// TIA Portal V17 export
// export: Created 2026-04-13T11:12:44.4398568Z, ExportSetting WithDefaults, DisplayName Totally Integrated Automation Portal, DisplayVersion V17 Update 4, DisplayName TIA Portal Openness, DisplayVersion V17 Update 4, DisplayName TIA Portal Version Control Interface, DisplayVersion V17, DisplayName SINAMICS Startdrive Advanced, DisplayVersion V17, DisplayName SINAMICS Startdrive G130, G150, S120, S150, SINAMICS MV, S210, DisplayVersion V17, DisplayName SINAMICS Startdrive G110M, G120, G120C, G120D, G120P, G115D, DisplayVersion V17, DisplayName STEP 7 Professional, DisplayVersion V17 Update 4, DisplayName STEP 7 Safety, DisplayVersion V17, DisplayName WinCC Professional, DisplayVersion V17 Update 4
DATA_BLOCK "6-ALLALARM_DB"   // DB23
VERSION : 0.1
// stored: AutoNumber true, DBAccessibleFromOPCUA true, DBAccessibleFromWebserver true, InstanceOfName B1--ALARM, InstanceOfType FB
"B1--ALARM"
   // VAR
   //    报警列表1 { S7_SetPoint := 'True'} : "A8-报警功能块";
   //    报警列表2 { S7_SetPoint := 'True'} : "A8-报警功能块";
   //    报警列表3 { S7_SetPoint := 'True'} : "A8-报警功能块";
   //    报警列表4 { S7_SetPoint := 'True'} : "A8-报警功能块";
   //    报警列表5 { S7_SetPoint := 'True'} : "A8-报警功能块";
   //    报警列表6 { S7_SetPoint := 'True'} : "A8-报警功能块";
   //    报警列表7 { S7_SetPoint := 'True'} : "A8-报警功能块";
   //    报警列表8 { S7_SetPoint := 'True'} : "A8-报警功能块";
   //    报警列表9 { S7_SetPoint := 'True'} : "A8-报警功能块";
   //    报警列表10 { S7_SetPoint := 'True'} : "A8-报警功能块";
   //    报警列表11 { S7_SetPoint := 'True'} : "A8-报警功能块";
   //    报警列表12 { S7_SetPoint := 'True'} : "A8-报警功能块";
   //    报警列表13 { S7_SetPoint := 'True'} : "A8-报警功能块";
   // END_VAR
BEGIN
END_DATA_BLOCK
